INTERFACE IRandom

/// Returns the next random variable
METHOD Next : LREAL
END_METHOD

METHOD SetSeed
VAR_INPUT
  seed : INT;
END_VAR
END_METHOD

END_INTERFACE

(* stored: Version 1.1.0.1, ProductVersion 3.1.4024.9
   Itf IRandom: Id {40ab6b77-e8c8-46c2-aa45-71150d6fb8b1}
   Method Next: Id {0bd8e0e8-7498-48a4-be55-845cfcc9e131}
   Method SetSeed: Id {874775a6-aa07-4087-9b58-128db7f5fca4} *)
